ABB RobotStudio station: SmartComponent dev.rsstnx

Station SmartComponent dev (saved by RobotStudio 25.1.11133.0)
Controller IRB1100_4_58, task T_ROB1: task frame (RAPID world) sits at (0, 0, 0) mm, rotated rx 0 ry 0 rz -90 deg in the station
Controller IRB1100_4_58
  mechanical unit ROB_1: IRB1100_4_58__02, 6 joints, base frame (0, 0, 0) mm
Layout (positions relative to the parent item):
  - IRB1100_4_58__02 [mechanism, from %ABB.RobotStudio.Models.IRB1100%\IRB1100_4_58__02.rslib] at (0, 0, 0) mm, rotated rx 0 ry 0 rz -90 deg; joint values [0, 0, 0, 0, 0.5236, 0] (rad or m)
  - SmartComponent_1 [smart component]
      signals: DI turnCONVEYORon
      connections:
        SmartComponent_1.turnCONVEYORon -> Highlighter.Active
    - Highlighter [smart component, from Components\Highlighter.rslib]
        properties: Object=950_4000_h2; Color=[0 204 0]; Opacity=255
  - 950_4000_h2 [part, from %ABB.RobotStudio.Models.Conveyors%\Conveyor 950 4000 h2.rslib] at (772.39, 0, 0) mm
Station logic (signal -> signal, property => property):
  IRB1100_4_58.ChangeColor -> SmartComponent_1.turnCONVEYORon
